FUNCTION_BLOCK FB_Machine
VAR_INPUT
END_VAR
VAR_OUTPUT
END_VAR
VAR
	fbUnit : ARRAY[0..MAX_UNIT_NUMBER - 1] OF FB_Unit;
	NumberOfUnit : BYTE := MAX_UNIT_NUMBER;
	oldNumberOfUnit : BYTE;
	Command : E_Command;
	GenerateCommand : E_Command;
	oldCommand : E_Command;
	
	fbLED : ARRAY[0..MAX_UNIT_NUMBER - 1] OF FB_LED;
	ledIndex : BYTE;
	CurrentUnitNum : INT;
	NextUnitNum			:	INT;
	LEDLocation			:	ARRAY[1..2] OF INT;

	i : BYTE;
	binit : BOOL;
	bButtonInit : BOOL;
	
	ForwardButton : FB_Button;
	BackwardButton : FB_Button;
	StopButton : FB_Button;
	GenerateButton : FB_Button;
END_VAR

ButtonLogic();
IF oldNumberOfUnit <> NumberOfUnit  THEN
	bInit := FALSE;
	ledIndex := 0;
	FOR i:= 0 TO MAX_UNIT_NUMBER - 1 BY 1 DO
		fbLED[i].Reset();
	END_FOR
END_IF

IF isCommandDirectionChanged THEN 
	bInit := FALSE;
END_IF
oldCommand := Command;
oldNumberOfUnit := NumberOfUnit;

IF NOT bInit THEN
	Initalize();
END_IF

GenerateLogic();

(* It assign Unit Interfaces for FB_LED *)
FOR i:= 0 TO MAX_UNIT_NUMBER - 1 BY 1 DO
	IF Command = E_Command.Forward THEN
		CurrentUnitNum := fbLED[i].Location1/5;
		NextUnitNum := fbLED[i].Location1/5 + 1;
		IF NextUnitNum >= MAX_UNIT_NUMBER THEN
			fbLED[i].GetFB_Unit(fbUnit[CurrentUnitNum], 0);
			CONTINUE;
		END_IF
		fbLED[i].GetFB_Unit(fbUnit[CurrentUnitNum], fbUnit[NextUnitNum]);
	ELSIF Command = E_Command.Backward THEN
		CurrentUnitNum := fbLED[i].Location2/5;
		NextUnitNum := fbLED[i].Location2/5 - 1;
		IF NextUnitNum < 0 THEN
			fbLED[i].GetFB_Unit(fbUnit[CurrentUnitNum], 0);
			CONTINUE;
		END_IF
		fbLED[i].GetFB_Unit(fbUnit[CurrentUnitNum], fbUnit[NextUnitNum]);
	END_IF
END_FOR

(* LED Control *)
FOR i:= 0 TO MAX_UNIT_NUMBER - 1 BY 1 DO
	fbUnit[i]();
END_FOR
FOR i:=0 TO ledIndex BY 1 DO
	IF fbLED[i].Location1 = -1 OR fbLED[i].Location2 = -1 THEN
		CONTINUE;
	END_IF
	LEDLocation[1] := fbLED[i].Location1;
	fbUnit[LEDLocation[1]/5].TurnOnLED(LEDLocation[1] MOD 5);
	LEDLocation[2] := fbLED[i].Location2;
	fbUnit[LEDLocation[2]/5].TurnOnLED(LEDLocation[2] MOD 5);
END_FOR
FOR i:= 0 TO MAX_UNIT_NUMBER - 1 BY 1 DO
	fbUnit[i].UpdateStatus();
END_FOR
FOR i:= 0 TO MAX_UNIT_NUMBER - 1 BY 1 DO
	fbLED[i]();
END_FOR

METHOD PRIVATE ButtonLogic : BOOL
VAR_INPUT
END_VAR
IF NOT bButtonInit THEN
	ForwardButton.Initalize(command, E_Command.Forward);
	BackwardButton.Initalize(command, E_Command.Backward);
	StopButton.Initalize(command, E_Command.Stop);
	GenerateButton.Initalize(GenerateCommand, E_Command.Generate);
	bButtonInit := TRUE;
	RETURN;
END_IF

ForwardButton();
BackwardButton();
StopButton();
GenerateButton();
END_METHOD

PROPERTY FirstUnitNumber : INT
GET
//IF Command = E_Command.Forward THEN
//	FirstUnitNumber := 0;
IF Command = E_Command.Backward THEN
	FirstUnitNumber := MAX_UNIT_NUMBER - 1;
ELSE
	FirstUnitNumber := 0;
END_IF
END_GET
END_PROPERTY

METHOD PRIVATE GenerateLogic
VAR_INPUT
END_VAR
IF GenerateCommand = E_Command.Generate AND fbUnit[0].isReceiveable THEN
	fbLED[ledIndex].Initalize(Command);
	ledIndex := ledIndex + 1;
	GenerateCommand := E_Command.Stop;
	ledIndex := LIMIT(0,ledIndex,MAX_UNIT_NUMBER - 1);
ELSE
	GenerateCommand := E_Command.Stop;
END_IF
END_METHOD

METHOD Initalize : BOOL
VAR_INPUT
END_VAR
NumberOfUnit := LIMIT(1,NumberOfUnit,MAX_UNIT_NUMBER);
FOR i:= 0 TO MAX_UNIT_NUMBER - 1 BY 1 DO
	fbUnit[i].Initalize(Command, i, 0, 0);
END_FOR

IF Command = E_Command.Forward THEN
	fbUnit[0].Initalize(Command, 0, 0, fbUnit[1]);
	FOR i:= 1 TO NumberOfUnit - 2 BY 1 DO
		fbUnit[i].Initalize(Command, i, fbUnit[i-1], fbUnit[i+1]);
	END_FOR
	fbUnit[NumberOfUnit - 1].Initalize(Command, NumberOfUnit-2, fbUnit[NumberOfUnit -2 ], 0);
ELSIF Command = E_Command.Backward THEN
	fbUnit[NumberOfUnit -1 ].Initalize(Command, NumberOfUnit-2, 0, fbUnit[NumberOfUnit - 2]);
	FOR i:= NumberOfUnit - 2 TO  1 BY -1 DO
		fbUnit[i].Initalize(Command, i, fbUnit[i+1], fbUnit[i-1]);
	END_FOR
	fbUnit[0].Initalize(Command, 0, fbUnit[1], 0);
END_IF

bInit := TRUE;
END_METHOD

PROPERTY isCommandDirectionChanged : BOOL
GET
isCommandDirectionChanged := (Command = E_Command.Forward AND oldCommand = E_Command.Backward) OR (Command = E_Command.Backward AND oldCommand = E_Command.Forward);
END_GET
END_PROPERTY

PROPERTY LastUnitNumber : INT
GET
//IF Command = E_Command.Forward THEN
//	LastUnitNumber := MAX_UNIT_NUMBER - 1;
IF Command = E_Command.Backward THEN
	LastUnitNumber := 0;
ELSE
	LastUnitNumber := MAX_UNIT_NUMBER - 1;
END_IF
END_GET
END_PROPERTY

END_FUNCTION_BLOCK

(* stored: Version 1.1.0.1, ProductVersion 3.1.4024.12
   POU FB_Machine: Id {f454b1e6-20f5-4637-accf-f47026bfc69d}, SpecialFunc None
   Method ButtonLogic: Id {bcb08168-26c3-45ec-8487-4274a995936e}
   Property FirstUnitNumber: Id {00651eac-699c-4216-aac1-8be740748c51}
   Get Get: Id {1df55a05-c3a7-4064-8953-e0289aec86ac}
   Method GenerateLogic: Id {117b607c-f975-4134-a958-56a2899754b8}
   Method Initalize: Id {a40c86fa-537a-421f-be3e-1fdb97d67ff4}
   Property isCommandDirectionChanged: Id {1de85dab-f228-4c9e-b46d-fa80c9045c50}
   Get Get: Id {1162b701-11e1-4463-9467-02d2d2714ad4}
   Property LastUnitNumber: Id {5808c0cf-5667-4f69-ac1d-42a16c95fad2}
   Get Get: Id {397cf324-af5b-4039-8c2a-f1a280514e55} *)
